FUNCTION_BLOCK FB_MotionVirtualFrame_Test EXTENDS TcUnit.FB_TestSuite
VAR
    nTestIDAssigner : INT;
    nTestID : INT := 1;
    tonTimeout : TON;
    tonStart : TON;

    stMotionStageRx : ST_MotionStage;
    stMotionStageRy : ST_MotionStage;
    stMotionStageRz : ST_MotionStage;

    stMotionStageVx : ST_MotionStage;
    stMotionStageVy : ST_MotionStage;
    stMotionStageVz : ST_MotionStage;

    fbMotionStageRx : FB_MotionStage;
    fbMotionStageRy : FB_MotionStage;
    fbMotionStageRz : FB_MotionStage;

    fbMotionStageVx : FB_MotionStage;
    fbMotionStageVy : FB_MotionStage;
    fbMotionStageVz : FB_MotionStage;

    nPositionCountsVx AT %Q* : UDINT;
    nPositionCountsVy AT %Q* : UDINT;
    nPositionCountsVz AT %Q* : UDINT;

    fbMotorTestSuite : FB_MotorTestSuite;
    fbMotionStageSetAndMoveHelper : FB_MotionStageSetAndMoveHelper;
    fbMotionStageSetHelperRx : FB_MotionStageSetHelper;
    fbMotionStageSetHelperRy : FB_MotionStageSetHelper;
    fbMotionStageSetHelperRz : FB_MotionStageSetHelper;
    fbMotionStageSetHelperVx : FB_MotionStageSetHelper;
    fbMotionStageSetHelperVy : FB_MotionStageSetHelper;
    fbMotionStageSetHelperVz : FB_MotionStageSetHelper;
    fbMotionVirtualFrame : FB_MotionVirtualFrame;
END_VAR


nTestIDAssigner := 0;

tonStart(IN := TRUE, PT := T#1s);

TestEnabled000045XYZMoveVxExpectNoErrorsCorrectPosVelAcc();

TestEnabled000090XYZMoveVxExpectNoErrorsCorrectPosVelAcc();

TestEnabled009090XYZMoveVxExpectNoErrorsCorrectPosVelAcc();

TestEnabled909090XYZMoveVxExpectNoErrorsCorrectPosVelAcc();

TestEnabledN22N21P4XYZMoveVxVyVzExpectNoErrorsCorrectPosVelAcc();

TestEnabledN22N21P4XYZMoveVyExpectNoErrorsCorrectPosVelAcc();

ACTION AssertNoErrors:

AssertFalse(
    Condition := tonTimeout.Q,
    Message := 'Timeout timer ended the test because it took longer than expected.'
);

AssertFalse(
    Condition := stMotionStageRx.bError,
    Message := 'Rx axis error detected when it should not have an error.'
);

AssertFalse(
    Condition := stMotionStageRy.bError,
    Message := 'Ry axis error detected when it should not have an error.'
);

AssertFalse(
    Condition := stMotionStageRz.bError,
    Message := 'Rz axis error detected when it should not have an error.'
);

AssertFalse(
    Condition := stMotionStageVx.bError,
    Message := 'Vx axis error detected when it should not have an error.'
);

AssertFalse(
    Condition := stMotionStageVy.bError,
    Message := 'Vy axis error detected when it should not have an error.'
);

AssertFalse(
    Condition := stMotionStageVz.bError,
    Message := 'Vz axis error detected when it should not have an error.'
);
END_ACTION


METHOD PRIVATE AssertPosVelAccCorrect
VAR_INPUT
    fDelta : LREAL;

    fRxPosExpected : LREAL;
    fRyPosExpected : LREAL;
    fRzPosExpected : LREAL;
    fVxPosExpected : LREAL;
    fVyPosExpected : LREAL;
    fVzPosExpected : LREAL;

    fRxVelExpected : LREAL;
    fRyVelExpected : LREAL;
    fRzVelExpected : LREAL;
    fVxVelExpected : LREAL;
    fVyVelExpected : LREAL;
    fVzVelExpected : LREAL;

    fRxAccExpected : LREAL;
    fRyAccExpected : LREAL;
    fRzAccExpected : LREAL;
    fVxAccExpected : LREAL;
    fVyAccExpected : LREAL;
    fVzAccExpected : LREAL;
END_VAR

// Position
AssertEquals_LREAL(
    Expected := fRxPosExpected,
    Actual := stMotionStageRx.Axis.NcToPlc.ActPos,
    Delta := fDelta,
    Message := 'Rx did not end at expected position.'
);

AssertEquals_LREAL(
    Expected := fRyPosExpected,
    Actual := stMotionStageRy.Axis.NcToPlc.ActPos,
    Delta := fDelta,
    Message := 'Ry did not end at expected position.'
);

AssertEquals_LREAL(
    Expected := fRzPosExpected,
    Actual := stMotionStageRz.Axis.NcToPlc.ActPos,
    Delta := fDelta,
    Message := 'Rz did not end at expected position.'
);

AssertEquals_LREAL(
    Expected := fVxPosExpected,
    Actual := stMotionStageVx.Axis.NcToPlc.ActPos,
    Delta := fDelta,
    Message := 'Vx did not end at expected position.'
);

AssertEquals_LREAL(
    Expected := fVyPosExpected,
    Actual := stMotionStageVy.Axis.NcToPlc.ActPos,
    Delta := fDelta,
    Message := 'Vy did not end at expected position.'
);

AssertEquals_LREAL(
    Expected := fVzPosExpected,
    Actual := stMotionStageVz.Axis.NcToPlc.ActPos,
    Delta := fDelta,
    Message := 'Vz did not end at expected position.'
);

// Velocity
AssertEquals_LREAL(
    Expected := fRxVelExpected,
    Actual := stMotionStageRx.fVelocity,
    Delta := fDelta,
    Message := 'Rx did not use the expected velocity.'
);

AssertEquals_LREAL(
    Expected := fRyVelExpected,
    Actual := stMotionStageRy.fVelocity,
    Delta := fDelta,
    Message := 'Ry did not use the expected velocity.'
);

AssertEquals_LREAL(
    Expected := fRzVelExpected,
    Actual := stMotionStageRz.fVelocity,
    Delta := fDelta,
    Message := 'Rz did not use the expected velocity.'
);

AssertEquals_LREAL(
    Expected := fVxVelExpected,
    Actual := stMotionStageVx.fVelocity,
    Delta := fDelta,
    Message := 'Vx did not use the expected velocity.'
);

AssertEquals_LREAL(
    Expected := fVyVelExpected,
    Actual := stMotionStageVy.fVelocity,
    Delta := fDelta,
    Message := 'Vy did not use the expected velocity.'
);

AssertEquals_LREAL(
    Expected := fVzVelExpected,
    Actual := stMotionStageVz.fVelocity,
    Delta := fDelta,
    Message := 'Vz did not use the expected velocity.'
);

// Acceleration
AssertEquals_LREAL(
    Expected := fRxAccExpected,
    Actual := stMotionStageRx.fAcceleration,
    Delta := fDelta,
    Message := 'Rx did not use the expected acceleration.'
);

AssertEquals_LREAL(
    Expected := fRyAccExpected,
    Actual := stMotionStageRy.fAcceleration,
    Delta := fDelta,
    Message := 'Ry did not use the expected acceleration.'
);

AssertEquals_LREAL(
    Expected := fRzAccExpected,
    Actual := stMotionStageRz.fAcceleration,
    Delta := fDelta,
    Message := 'Rz did not use the expected acceleration.'
);

AssertEquals_LREAL(
    Expected := fVxAccExpected,
    Actual := stMotionStageVx.fAcceleration,
    Delta := fDelta,
    Message := 'Vx did not use the expected acceleration.'
);

AssertEquals_LREAL(
    Expected := fVyAccExpected,
    Actual := stMotionStageVy.fAcceleration,
    Delta := fDelta,
    Message := 'Vy did not use the expected acceleration.'
);

AssertEquals_LREAL(
    Expected := fVzAccExpected,
    Actual := stMotionStageVz.fAcceleration,
    Delta := fDelta,
    Message := 'Vz did not use the expected acceleration.'
);
END_METHOD


METHOD PRIVATE InitMotors : BOOL

fbMotorTestSuite.SetEnables(stMotionStage := stMotionStageRx);
fbMotorTestSuite.SetEnables(stMotionStage := stMotionStageRy);
fbMotorTestSuite.SetEnables(stMotionStage := stMotionStageRz);
fbMotorTestSuite.SetEnables(stMotionStage := stMotionStageVx);
fbMotorTestSuite.SetEnables(stMotionStage := stMotionStageVy);
fbMotorTestSuite.SetEnables(stMotionStage := stMotionStageVz);

SetTar0();

fbMotionStageSetHelperRx(
    bExecute := TRUE,
    fStartPosition := 0.0,
    stMotionStage := stMotionStageRx,
    bResetDone => ,
    bSetDone =>
);

fbMotionStageSetHelperRy(
    bExecute := TRUE,
    fStartPosition := 0.0,
    stMotionStage := stMotionStageRy,
    bResetDone => ,
    bSetDone =>
);

fbMotionStageSetHelperRz(
    bExecute := TRUE,
    fStartPosition := 0.0,
    stMotionStage := stMotionStageRz,
    bResetDone => ,
    bSetDone =>
);

fbMotionStageSetHelperVx(
    bExecute := TRUE,
    fStartPosition := 0.0,
    stMotionStage := stMotionStageVx,
    bResetDone => ,
    bSetDone =>
);

fbMotionStageSetHelperVy(
    bExecute := TRUE,
    fStartPosition := 0.0,
    stMotionStage := stMotionStageVy,
    bResetDone => ,
    bSetDone =>
);

fbMotionStageSetHelperVz(
    bExecute := TRUE,
    fStartPosition := 0.0,
    stMotionStage := stMotionStageVz,
    bResetDone => ,
    bSetDone =>
);

IF fbMotionStageSetHelperRx.bSetDone AND
   fbMotionStageSetHelperRy.bSetDone AND
   fbMotionStageSetHelperRz.bSetDone AND
   fbMotionStageSetHelperVx.bSetDone AND
   fbMotionStageSetHelperVy.bSetDone AND
   fbMotionStageSetHelperVz.bSetDone THEN

    fbMotionStageSetHelperRx(
        bExecute := FALSE,
        fStartPosition := 0.0,
        stMotionStage := stMotionStageRx,
        bResetDone => ,
        bSetDone =>
    );

    fbMotionStageSetHelperRy(
        bExecute := FALSE,
        fStartPosition := 0.0,
        stMotionStage := stMotionStageRy,
        bResetDone => ,
        bSetDone =>
    );

    fbMotionStageSetHelperRz(
        bExecute := FALSE,
        fStartPosition := 0.0,
        stMotionStage := stMotionStageRz,
        bResetDone => ,
        bSetDone =>
    );

    fbMotionStageSetHelperVx(
        bExecute := FALSE,
        fStartPosition := 0.0,
        stMotionStage := stMotionStageVx,
        bResetDone => ,
        bSetDone =>
    );

    fbMotionStageSetHelperVy(
        bExecute := FALSE,
        fStartPosition := 0.0,
        stMotionStage := stMotionStageVy,
        bResetDone => ,
        bSetDone =>
    );

    fbMotionStageSetHelperVz(
        bExecute := FALSE,
        fStartPosition := 0.0,
        stMotionStage := stMotionStageVz,
        bResetDone => ,
        bSetDone =>
    );

    stMotionStageRx.nEnableMode := E_StageEnableMode.ALWAYS;
    stMotionStageRy.nEnableMode := E_StageEnableMode.ALWAYS;
    stMotionStageRz.nEnableMode := E_StageEnableMode.ALWAYS;
    stMotionStageVx.nEnableMode := E_StageEnableMode.ALWAYS;
    stMotionStageVy.nEnableMode := E_StageEnableMode.ALWAYS;
    stMotionStageVz.nEnableMode := E_StageEnableMode.ALWAYS;

    IF stMotionStageRx.bAllEnable AND
        stMotionStageRy.bAllEnable AND
        stMotionStageRz.bAllEnable AND
        stMotionStageVx.bAllEnable AND
        stMotionStageVy.bAllEnable AND
        stMotionStageVz.bAllEnable THEN

        InitMotors := TRUE;
    END_IF
END_IF
END_METHOD


METHOD PRIVATE SetTar0

stMotionStageVx.fPosition := 0.0;
stMotionStageVx.fVelocity := 0.0;
stMotionStageVx.fAcceleration := 0.0;

stMotionStageVy.fPosition := 0.0;
stMotionStageVy.fVelocity := 0.0;
stMotionStageVy.fAcceleration := 0.0;

stMotionStageVz.fPosition := 0.0;
stMotionStageVz.fVelocity := 0.0;
stMotionStageVz.fAcceleration := 0.0;

stMotionStageRx.fPosition := 0.0;
stMotionStageRx.fVelocity := 0.0;
stMotionStageRx.fAcceleration := 0.0;

stMotionStageRy.fPosition := 0.0;
stMotionStageRy.fVelocity := 0.0;
stMotionStageRy.fAcceleration := 0.0;

stMotionStageRz.fPosition := 0.0;
stMotionStageRz.fVelocity := 0.0;
stMotionStageRz.fAcceleration := 0.0;
END_METHOD


METHOD PRIVATE TestEnabled000045XYZMoveVxExpectNoErrorsCorrectPosVelAcc
VAR_INST
    bInit : BOOL;
    bComplete : BOOL;
    bBusyReached : BOOL;
    rtMoveCmdOnce : R_TRIG;
    fDelta : LREAL := 1e-9;
END_VAR

TEST('TestEnabled000045XYZMoveVxExpectNoErrorsCorrectPosVelAcc');

nTestIDAssigner := nTestIDAssigner + 1;

IF nTestID <> nTestIDAssigner OR NOT tonStart.Q THEN
    RETURN;
END_IF

tonTimeout(IN := TRUE, PT := T#3s);

IF NOT bInit THEN
    bInit := InitMotors();
END_IF

IF bInit THEN
    stMotionStageVx.fPosition := 15.0;
    stMotionStageVx.fVelocity := stMotionStageVx.fPosition * 2.0 / 3.0;
    stMotionStageVx.fAcceleration := stMotionStageVx.fVelocity * 5.0;
    rtMoveCmdOnce(CLK := TRUE);
    stMotionStageVx.bMoveCmd := rtMoveCmdOnce.Q;
END_IF

fbMotionVirtualFrame(
    stMotionStageRx := stMotionStageRx,
    stMotionStageRy := stMotionStageRy,
    stMotionStageRz := stMotionStageRz,
    stMotionStageVx := stMotionStageVx,
    stMotionStageVy := stMotionStageVy,
    stMotionStageVz := stMotionStageVz,
    bEnable := TRUE,
    fAlphaDegrees := 0.0,
    fBetaDegrees := 0.0,
    fGammaDegrees := 45.0,
    sOrder := 'XYZ',
    bBaseToNew := TRUE,
    fbVirtActPositionVec3 => ,
    fbVirtActVelocityVec3 => ,
    fbVirtActAcceleraVec3 =>
);

IF stMotionStageVx.bBusy THEN
    bBusyReached := TRUE;
END_IF

IF bBusyReached AND NOT stMotionStageVx.bBusy THEN
    bComplete := TRUE;
END_IF

IF (bComplete AND
    NOT stMotionStageVx.bBusy AND
    NOT stMotionStageVy.bBusy AND
    NOT stMotionStageVz.bBusy AND
    NOT stMotionStageRx.bBusy AND
    NOT stMotionStageRy.bBusy AND
    NOT stMotionStageRz.bBusy)
    OR tonTimeout.Q THEN

    AssertNoErrors();

    AssertPosVelAccCorrect(
        fDelta := fDelta,
        fRxPosExpected := stMotionStageVx.fPosition * SQRT(2.0) / 2.0,
        fRyPosExpected := stMotionStageVx.fPosition * SQRT(2.0) / 2.0,
        fRzPosExpected := 0.0,
        fVxPosExpected := stMotionStageVx.fPosition,
        fVyPosExpected := 0.0,
        fVzPosExpected := 0.0,
        fRxVelExpected := stMotionStageVx.fVelocity * SQRT(2.0) / 2.0,
        fRyVelExpected := stMotionStageVx.fVelocity * SQRT(2.0) / 2.0,
        fRzVelExpected := 0.0,
        fVxVelExpected := stMotionStageVx.fVelocity,
        fVyVelExpected := 0.0,
        fVzVelExpected := 0.0,
        fRxAccExpected := stMotionStageVx.fAcceleration * SQRT(2.0) / 2.0,
        fRyAccExpected := stMotionStageVx.fAcceleration * SQRT(2.0) / 2.0,
        fRzAccExpected := 0.0,
        fVxAccExpected := stMotionStageVx.fAcceleration,
        fVyAccExpected := 0.0,
        fVzAccExpected := 0.0
    );

    TEST_FINISHED();

    tonTimeout(IN := FALSE);

    nTestID := nTestID + 1;
END_IF

fbMotionStageRx(stMotionStage := stMotionStageRx);
fbMotionStageRy(stMotionStage := stMotionStageRy);
fbMotionStageRz(stMotionStage := stMotionStageRz);

fbMotionStageVx(stMotionStage := stMotionStageVx);
fbMotionStageVy(stMotionStage := stMotionStageVy);
fbMotionStageVz(stMotionStage := stMotionStageVz);

nPositionCountsVx := LREAL_TO_UDINT((fbMotionVirtualFrame.fbVirtActPositionVec3.x + 100.0) * 1e6);
nPositionCountsVy := LREAL_TO_UDINT((fbMotionVirtualFrame.fbVirtActPositionVec3.y + 100.0) * 1e6);
nPositionCountsVz := LREAL_TO_UDINT((fbMotionVirtualFrame.fbVirtActPositionVec3.z + 100.0) * 1e6);
END_METHOD


METHOD PRIVATE TestEnabled000090XYZMoveVxExpectNoErrorsCorrectPosVelAcc
VAR_INST
    bInit : BOOL;
    bComplete : BOOL;
    bBusyReached : BOOL;
    rtMoveCmdOnce : R_TRIG;
    fDelta : LREAL := 1e-9;
END_VAR

TEST('TestEnabled000090XYZMoveVxExpectNoErrorsCorrectPosVelAcc');

nTestIDAssigner := nTestIDAssigner + 1;

IF nTestID <> nTestIDAssigner OR NOT tonStart.Q THEN
    RETURN;
END_IF

tonTimeout(IN := TRUE, PT := T#3s);

IF NOT bInit THEN
    bInit := InitMotors();
END_IF

IF bInit THEN
    stMotionStageVx.fPosition := 20.0;
    stMotionStageVx.fVelocity := stMotionStageVx.fPosition * 2.0 / 3.0;
    stMotionStageVx.fAcceleration := stMotionStageVx.fVelocity * 5.0;
    rtMoveCmdOnce(CLK := TRUE);
    stMotionStageVx.bMoveCmd := rtMoveCmdOnce.Q;
END_IF

fbMotionVirtualFrame(
    stMotionStageRx := stMotionStageRx,
    stMotionStageRy := stMotionStageRy,
    stMotionStageRz := stMotionStageRz,
    stMotionStageVx := stMotionStageVx,
    stMotionStageVy := stMotionStageVy,
    stMotionStageVz := stMotionStageVz,
    bEnable := TRUE,
    fAlphaDegrees := 0.0,
    fBetaDegrees := 0.0,
    fGammaDegrees := 90.0,
    sOrder := 'XYZ',
    bBaseToNew := TRUE,
    fbVirtActPositionVec3 => ,
    fbVirtActVelocityVec3 => ,
    fbVirtActAcceleraVec3 =>
);

IF stMotionStageVx.bBusy THEN
    bBusyReached := TRUE;
END_IF

IF bBusyReached AND NOT stMotionStageVx.bBusy THEN
    bComplete := TRUE;
END_IF

IF (bComplete AND
    NOT stMotionStageVx.bBusy AND
    NOT stMotionStageVy.bBusy AND
    NOT stMotionStageVz.bBusy AND
    NOT stMotionStageRx.bBusy AND
    NOT stMotionStageRy.bBusy AND
    NOT stMotionStageRz.bBusy)
    OR tonTimeout.Q THEN

    AssertNoErrors();

    AssertPosVelAccCorrect(
        fDelta := fDelta,
        fRxPosExpected := 0.0,
        fRyPosExpected := stMotionStageVx.fPosition,
        fRzPosExpected := 0.0,
        fVxPosExpected := stMotionStageVx.fPosition,
        fVyPosExpected := 0.0,
        fVzPosExpected := 0.0,
        fRxVelExpected := 0.0,
        fRyVelExpected := stMotionStageVx.fVelocity,
        fRzVelExpected := 0.0,
        fVxVelExpected := stMotionStageVx.fVelocity,
        fVyVelExpected := 0.0,
        fVzVelExpected := 0.0,
        fRxAccExpected := 0.0,
        fRyAccExpected := stMotionStageVx.fAcceleration,
        fRzAccExpected := 0.0,
        fVxAccExpected := stMotionStageVx.fAcceleration,
        fVyAccExpected := 0.0,
        fVzAccExpected := 0.0
    );

    TEST_FINISHED();

    tonTimeout(IN := FALSE);

    nTestID := nTestID + 1;
END_IF

fbMotionStageRx(stMotionStage := stMotionStageRx);
fbMotionStageRy(stMotionStage := stMotionStageRy);
fbMotionStageRz(stMotionStage := stMotionStageRz);

fbMotionStageVx(stMotionStage := stMotionStageVx);
fbMotionStageVy(stMotionStage := stMotionStageVy);
fbMotionStageVz(stMotionStage := stMotionStageVz);

nPositionCountsVx := LREAL_TO_UDINT((fbMotionVirtualFrame.fbVirtActPositionVec3.x + 100.0) * 1e6);
nPositionCountsVy := LREAL_TO_UDINT((fbMotionVirtualFrame.fbVirtActPositionVec3.y + 100.0) * 1e6);
nPositionCountsVz := LREAL_TO_UDINT((fbMotionVirtualFrame.fbVirtActPositionVec3.z + 100.0) * 1e6);
END_METHOD


METHOD PRIVATE TestEnabled009090XYZMoveVxExpectNoErrorsCorrectPosVelAcc
VAR_INST
    bInit : BOOL;
    bComplete : BOOL;
    bBusyReached : BOOL;
    rtMoveCmdOnce : R_TRIG;
    fDelta : LREAL := 1e-9;
END_VAR

TEST('TestEnabled009090XYZMoveVxExpectNoErrorsCorrectPosVelAcc');

nTestIDAssigner := nTestIDAssigner + 1;

IF nTestID <> nTestIDAssigner OR NOT tonStart.Q THEN
    RETURN;
END_IF

tonTimeout(IN := TRUE, PT := T#3s);

IF NOT bInit THEN
    bInit := InitMotors();
END_IF

IF bInit THEN
    stMotionStageVx.fPosition := 25.0;
    stMotionStageVx.fVelocity := stMotionStageVx.fPosition * 2.0 / 3.0;
    stMotionStageVx.fAcceleration := stMotionStageVx.fVelocity * 5.0;
    rtMoveCmdOnce(CLK := TRUE);
    stMotionStageVx.bMoveCmd := rtMoveCmdOnce.Q;
END_IF

fbMotionVirtualFrame(
    stMotionStageRx := stMotionStageRx,
    stMotionStageRy := stMotionStageRy,
    stMotionStageRz := stMotionStageRz,
    stMotionStageVx := stMotionStageVx,
    stMotionStageVy := stMotionStageVy,
    stMotionStageVz := stMotionStageVz,
    bEnable := TRUE,
    fAlphaDegrees := 0.0,
    fBetaDegrees := 90.0,
    fGammaDegrees := 90.0,
    sOrder := 'XYZ',
    bBaseToNew := TRUE,
    fbVirtActPositionVec3 => ,
    fbVirtActVelocityVec3 => ,
    fbVirtActAcceleraVec3 =>
);

IF stMotionStageVx.bBusy THEN
    bBusyReached := TRUE;
END_IF

IF bBusyReached AND NOT stMotionStageVx.bBusy THEN
    bComplete := TRUE;
END_IF

IF (bComplete AND
    NOT stMotionStageVx.bBusy AND
    NOT stMotionStageVy.bBusy AND
    NOT stMotionStageVz.bBusy AND
    NOT stMotionStageRx.bBusy AND
    NOT stMotionStageRy.bBusy AND
    NOT stMotionStageRz.bBusy)
    OR tonTimeout.Q THEN

    AssertNoErrors();

    AssertPosVelAccCorrect(
        fDelta := fDelta,
        fRxPosExpected := 0.0,
        fRyPosExpected := stMotionStageVx.fPosition,
        fRzPosExpected := 0.0,
        fVxPosExpected := stMotionStageVx.fPosition,
        fVyPosExpected := 0.0,
        fVzPosExpected := 0.0,
        fRxVelExpected := 0.0,
        fRyVelExpected := stMotionStageVx.fVelocity,
        fRzVelExpected := 0.0,
        fVxVelExpected := stMotionStageVx.fVelocity,
        fVyVelExpected := 0.0,
        fVzVelExpected := 0.0,
        fRxAccExpected := 0.0,
        fRyAccExpected := stMotionStageVx.fAcceleration,
        fRzAccExpected := 0.0,
        fVxAccExpected := stMotionStageVx.fAcceleration,
        fVyAccExpected := 0.0,
        fVzAccExpected := 0.0
    );

    TEST_FINISHED();

    tonTimeout(IN := FALSE);

    nTestID := nTestID + 1;
END_IF

fbMotionStageRx(stMotionStage := stMotionStageRx);
fbMotionStageRy(stMotionStage := stMotionStageRy);
fbMotionStageRz(stMotionStage := stMotionStageRz);

fbMotionStageVx(stMotionStage := stMotionStageVx);
fbMotionStageVy(stMotionStage := stMotionStageVy);
fbMotionStageVz(stMotionStage := stMotionStageVz);

nPositionCountsVx := LREAL_TO_UDINT((fbMotionVirtualFrame.fbVirtActPositionVec3.x + 100.0) * 1e6);
nPositionCountsVy := LREAL_TO_UDINT((fbMotionVirtualFrame.fbVirtActPositionVec3.y + 100.0) * 1e6);
nPositionCountsVz := LREAL_TO_UDINT((fbMotionVirtualFrame.fbVirtActPositionVec3.z + 100.0) * 1e6);
END_METHOD


METHOD PRIVATE TestEnabled909090XYZMoveVxExpectNoErrorsCorrectPosVelAcc
VAR_INST
    bInit : BOOL;
    bComplete : BOOL;
    bBusyReached : BOOL;
    rtMoveCmdOnce : R_TRIG;
    fDelta : LREAL := 1e-9;
END_VAR

TEST('TestEnabled909090XYZMoveVxExpectNoErrorsCorrectPosVelAcc');

nTestIDAssigner := nTestIDAssigner + 1;

IF nTestID <> nTestIDAssigner OR NOT tonStart.Q THEN
    RETURN;
END_IF

tonTimeout(IN := TRUE, PT := T#3s);

IF NOT bInit THEN
    bInit := InitMotors();
END_IF

IF bInit THEN
    stMotionStageVx.fPosition := 35.0;
    stMotionStageVx.fVelocity := stMotionStageVx.fPosition * 2.0 / 3.0;
    stMotionStageVx.fAcceleration := stMotionStageVx.fVelocity * 5.0;
    rtMoveCmdOnce(CLK := TRUE);
    stMotionStageVx.bMoveCmd := rtMoveCmdOnce.Q;
END_IF

fbMotionVirtualFrame(
    stMotionStageRx := stMotionStageRx,
    stMotionStageRy := stMotionStageRy,
    stMotionStageRz := stMotionStageRz,
    stMotionStageVx := stMotionStageVx,
    stMotionStageVy := stMotionStageVy,
    stMotionStageVz := stMotionStageVz,
    bEnable := TRUE,
    fAlphaDegrees := 90.0,
    fBetaDegrees := 90.0,
    fGammaDegrees := 90.0,
    sOrder := 'XYZ',
    bBaseToNew := TRUE,
    fbVirtActPositionVec3 => ,
    fbVirtActVelocityVec3 => ,
    fbVirtActAcceleraVec3 =>
);

IF stMotionStageVx.bBusy THEN
    bBusyReached := TRUE;
END_IF

IF bBusyReached AND NOT stMotionStageVx.bBusy THEN
    bComplete := TRUE;
END_IF

IF (bComplete AND
    NOT stMotionStageVx.bBusy AND
    NOT stMotionStageVy.bBusy AND
    NOT stMotionStageVz.bBusy AND
    NOT stMotionStageRx.bBusy AND
    NOT stMotionStageRy.bBusy AND
    NOT stMotionStageRz.bBusy)
    OR tonTimeout.Q THEN

    AssertNoErrors();

    AssertPosVelAccCorrect(
        fDelta := fDelta,
        fRxPosExpected := 0.0,
        fRyPosExpected := 0.0,
        fRzPosExpected := stMotionStageVx.fPosition,
        fVxPosExpected := stMotionStageVx.fPosition,
        fVyPosExpected := 0.0,
        fVzPosExpected := 0.0,
        fRxVelExpected := 0.0,
        fRyVelExpected := 0.0,
        fRzVelExpected := stMotionStageVx.fVelocity,
        fVxVelExpected := stMotionStageVx.fVelocity,
        fVyVelExpected := 0.0,
        fVzVelExpected := 0.0,
        fRxAccExpected := 0.0,
        fRyAccExpected := 0.0,
        fRzAccExpected := stMotionStageVx.fAcceleration,
        fVxAccExpected := stMotionStageVx.fAcceleration,
        fVyAccExpected := 0.0,
        fVzAccExpected := 0.0
    );

    TEST_FINISHED();

    tonTimeout(IN := FALSE);

    nTestID := nTestID + 1;
END_IF

fbMotionStageRx(stMotionStage := stMotionStageRx);
fbMotionStageRy(stMotionStage := stMotionStageRy);
fbMotionStageRz(stMotionStage := stMotionStageRz);

fbMotionStageVx(stMotionStage := stMotionStageVx);
fbMotionStageVy(stMotionStage := stMotionStageVy);
fbMotionStageVz(stMotionStage := stMotionStageVz);

nPositionCountsVx := LREAL_TO_UDINT((fbMotionVirtualFrame.fbVirtActPositionVec3.x + 100.0) * 1e6);
nPositionCountsVy := LREAL_TO_UDINT((fbMotionVirtualFrame.fbVirtActPositionVec3.y + 100.0) * 1e6);
nPositionCountsVz := LREAL_TO_UDINT((fbMotionVirtualFrame.fbVirtActPositionVec3.z + 100.0) * 1e6);
END_METHOD


METHOD PRIVATE TestEnabledN22N21P4XYZMoveVxVyVzExpectNoErrorsCorrectPosVelAcc
VAR_INST
    bInit : BOOL;
    bComplete : BOOL;
    bBusyReached : BOOL;
    rtMoveCmdOnce : R_TRIG;
    fDelta : LREAL := 1e-9;
END_VAR

TEST('TestEnabledN22N21P4XYZMoveVxVyVzExpectNoErrorsCorrectPosVelAcc');

nTestIDAssigner := nTestIDAssigner + 1;

IF nTestID <> nTestIDAssigner OR NOT tonStart.Q THEN
    RETURN;
END_IF

tonTimeout(IN := TRUE, PT := T#3s);

IF NOT bInit THEN
    bInit := InitMotors();
END_IF

IF bInit THEN
    rtMoveCmdOnce(CLK := TRUE);

    stMotionStageVx.fPosition := 15.0;
    stMotionStageVx.fVelocity := stMotionStageVx.fPosition * 2.0 / 3.0;
    stMotionStageVx.fAcceleration := stMotionStageVx.fVelocity * 5.0;
    stMotionStageVx.bMoveCmd := rtMoveCmdOnce.Q;

    stMotionStageVy.fPosition := -30.0;
    stMotionStageVy.fVelocity := ABS(stMotionStageVy.fPosition * 2.0 / 3.0);
    stMotionStageVy.fAcceleration := ABS(stMotionStageVy.fVelocity * 5.0);
    stMotionStageVy.bMoveCmd := rtMoveCmdOnce.Q;

    stMotionStageVz.fPosition := 45.0;
    stMotionStageVz.fVelocity := stMotionStageVz.fPosition * 2.0 / 3.0;
    stMotionStageVz.fAcceleration := stMotionStageVz.fVelocity * 5.0;
    stMotionStageVz.bMoveCmd := rtMoveCmdOnce.Q;
END_IF

fbMotionVirtualFrame(
    stMotionStageRx := stMotionStageRx,
    stMotionStageRy := stMotionStageRy,
    stMotionStageRz := stMotionStageRz,
    stMotionStageVx := stMotionStageVx,
    stMotionStageVy := stMotionStageVy,
    stMotionStageVz := stMotionStageVz,
    bEnable := TRUE,
    fAlphaDegrees := -22.21,
    fBetaDegrees := -20.7,
    fGammaDegrees := 3.793,
    sOrder := 'XYZ',
    bBaseToNew := FALSE,
    fbVirtActPositionVec3 => ,
    fbVirtActVelocityVec3 => ,
    fbVirtActAcceleraVec3 =>
);

IF stMotionStageVx.bBusy AND stMotionStageVy.bBusy AND stMotionStageVz.bBusy THEN
    bBusyReached := TRUE;
END_IF

IF bBusyReached AND NOT stMotionStageVx.bBusy AND NOT stMotionStageVy.bBusy AND NOT stMotionStageVz.bBusy THEN
    bComplete := TRUE;
END_IF

IF (bComplete AND
    NOT stMotionStageVx.bBusy AND
    NOT stMotionStageVy.bBusy AND
    NOT stMotionStageVz.bBusy AND
    NOT stMotionStageRx.bBusy AND
    NOT stMotionStageRy.bBusy AND
    NOT stMotionStageRz.bBusy)
    OR tonTimeout.Q THEN

    AssertNoErrors();

    AssertPosVelAccCorrect(
        fDelta := fDelta,
        fRxPosExpected := 21.732640182123049,
        fRyPosExpected := -46.323371856381527,
        fRzPosExpected := 23.061603816078627,
        fVxPosExpected := stMotionStageVx.fPosition,
        fVyPosExpected := stMotionStageVy.fPosition,
        fVzPosExpected := stMotionStageVz.fPosition,
        fRxVelExpected := 14.488426788082032,
        fRyVelExpected := 30.882247904254346,
        fRzVelExpected := 15.374402544052412,
        fVxVelExpected := stMotionStageVx.fVelocity,
        fVyVelExpected := stMotionStageVy.fVelocity,
        fVzVelExpected := stMotionStageVz.fVelocity,
        fRxAccExpected := 0.724421339404102 * 1e2,
        fRyAccExpected := 1.544112395212718 * 1e2,
        fRzAccExpected := 0.768720127202621 * 1e2,
        fVxAccExpected := stMotionStageVx.fAcceleration,
        fVyAccExpected := stMotionStageVy.fAcceleration,
        fVzAccExpected := stMotionStageVz.fAcceleration
    );

    TEST_FINISHED();

    tonTimeout(IN := FALSE);

    nTestID := nTestID + 1;
END_IF

fbMotionStageRx(stMotionStage := stMotionStageRx);
fbMotionStageRy(stMotionStage := stMotionStageRy);
fbMotionStageRz(stMotionStage := stMotionStageRz);

fbMotionStageVx(stMotionStage := stMotionStageVx);
fbMotionStageVy(stMotionStage := stMotionStageVy);
fbMotionStageVz(stMotionStage := stMotionStageVz);

nPositionCountsVx := LREAL_TO_UDINT((fbMotionVirtualFrame.fbVirtActPositionVec3.x + 100.0) * 1e6);
nPositionCountsVy := LREAL_TO_UDINT((fbMotionVirtualFrame.fbVirtActPositionVec3.y + 100.0) * 1e6);
nPositionCountsVz := LREAL_TO_UDINT((fbMotionVirtualFrame.fbVirtActPositionVec3.z + 100.0) * 1e6);
END_METHOD


METHOD PRIVATE TestEnabledN22N21P4XYZMoveVyExpectNoErrorsCorrectPosVelAcc
VAR_INST
    bInit : BOOL;
    bComplete : BOOL;
    bBusyReached : BOOL;
    rtMoveCmdOnce : R_TRIG;
    fDelta : LREAL := 1e-9;
END_VAR

TEST('TestEnabledN22N21P4XYZMoveVyExpectNoErrorsCorrectPosVelAcc');

nTestIDAssigner := nTestIDAssigner + 1;

IF nTestID <> nTestIDAssigner OR NOT tonStart.Q THEN
    RETURN;
END_IF

tonTimeout(IN := TRUE, PT := T#3s);

IF NOT bInit THEN
    bInit := InitMotors();
END_IF

IF bInit THEN
    stMotionStageVy.fPosition := 30.0;
    stMotionStageVy.fVelocity := stMotionStageVy.fPosition * 2.0 / 3.0;
    stMotionStageVy.fAcceleration := stMotionStageVy.fVelocity * 5.0;
    rtMoveCmdOnce(CLK := TRUE);
    stMotionStageVy.bMoveCmd := rtMoveCmdOnce.Q;
END_IF

fbMotionVirtualFrame(
    stMotionStageRx := stMotionStageRx,
    stMotionStageRy := stMotionStageRy,
    stMotionStageRz := stMotionStageRz,
    stMotionStageVx := stMotionStageVx,
    stMotionStageVy := stMotionStageVy,
    stMotionStageVz := stMotionStageVz,
    bEnable := TRUE,
    fAlphaDegrees := -22.21,
    fBetaDegrees := -20.7,
    fGammaDegrees := 3.793,
    sOrder := 'XYZ',
    bBaseToNew := FALSE,
    fbVirtActPositionVec3 => ,
    fbVirtActVelocityVec3 => ,
    fbVirtActAcceleraVec3 =>
);

IF stMotionStageVy.bBusy THEN
    bBusyReached := TRUE;
END_IF

IF bBusyReached AND NOT stMotionStageVy.bBusy THEN
    bComplete := TRUE;
END_IF

IF (bComplete AND
    NOT stMotionStageVx.bBusy AND
    NOT stMotionStageVy.bBusy AND
    NOT stMotionStageVz.bBusy AND
    NOT stMotionStageRx.bBusy AND
    NOT stMotionStageRy.bBusy AND
    NOT stMotionStageRz.bBusy)
    OR tonTimeout.Q THEN

    AssertNoErrors();

    AssertPosVelAccCorrect(
        fDelta := fDelta,
        fRxPosExpected := 5.836964390001455,
        fRyPosExpected := 27.448135465863341,
        fRzPosExpected := 10.608001987060069,
        fVxPosExpected := 0.0,
        fVyPosExpected := stMotionStageVy.fPosition,
        fVzPosExpected := 0.0,
        fRxVelExpected := 5.836964390001455 * 2.0 / 3.0,
        fRyVelExpected := 27.448135465863341 * 2.0 / 3.0,
        fRzVelExpected := 10.608001987060069 * 2.0 / 3.0,
        fVxVelExpected := 0.0,
        fVyVelExpected := stMotionStageVy.fVelocity,
        fVzVelExpected := 0.0,
        fRxAccExpected := 5.836964390001455 * 2.0 / 3.0 * 5.0,
        fRyAccExpected := 27.448135465863341 * 2.0 / 3.0 * 5.0,
        fRzAccExpected := 10.608001987060069 * 2.0 / 3.0 * 5.0,
        fVxAccExpected := 0.0,
        fVyAccExpected := stMotionStageVy.fAcceleration,
        fVzAccExpected := 0.0
    );

    TEST_FINISHED();

    tonTimeout(IN := FALSE);

    nTestID := nTestID + 1;
END_IF

fbMotionStageRx(stMotionStage := stMotionStageRx);
fbMotionStageRy(stMotionStage := stMotionStageRy);
fbMotionStageRz(stMotionStage := stMotionStageRz);

fbMotionStageVx(stMotionStage := stMotionStageVx);
fbMotionStageVy(stMotionStage := stMotionStageVy);
fbMotionStageVz(stMotionStage := stMotionStageVz);

nPositionCountsVx := LREAL_TO_UDINT((fbMotionVirtualFrame.fbVirtActPositionVec3.x + 100.0) * 1e6);
nPositionCountsVy := LREAL_TO_UDINT((fbMotionVirtualFrame.fbVirtActPositionVec3.y + 100.0) * 1e6);
nPositionCountsVz := LREAL_TO_UDINT((fbMotionVirtualFrame.fbVirtActPositionVec3.z + 100.0) * 1e6);
END_METHOD

END_FUNCTION_BLOCK

(* stored: Version 1.1.0.1
   POU FB_MotionVirtualFrame_Test: Id {89c3fcc0-8932-48a8-9976-db5e1ce2e9c1}, SpecialFunc None
   Action AssertNoErrors: Id {835be31f-8489-492c-bbc8-90f1a0c04eb1}
   Method AssertPosVelAccCorrect: Id {645a18f6-30c6-4966-a4ea-a55c7fe24cdb}
   Method InitMotors: Id {62a5dad0-d7c7-4660-a2ba-05b951ff6ec0}
   Method SetTar0: Id {46f058f5-eb38-4947-8a98-e9788bc7e851}
   Method TestEnabled000045XYZMoveVxExpectNoErrorsCorrectPosVelAcc: Id {2d40004f-479b-4cbc-9e82-633d171550b1}
   Method TestEnabled000090XYZMoveVxExpectNoErrorsCorrectPosVelAcc: Id {96619493-4949-4dca-ad6e-5a7f16038b00}
   Method TestEnabled009090XYZMoveVxExpectNoErrorsCorrectPosVelAcc: Id {1e6baa8a-c190-4123-9357-8013455bb605}
   Method TestEnabled909090XYZMoveVxExpectNoErrorsCorrectPosVelAcc: Id {6c8e3a8e-65f7-4fff-beca-5b108daa78c7}
   Method TestEnabledN22N21P4XYZMoveVxVyVzExpectNoErrorsCorrectPosVelAcc: Id {346202be-906d-4ffe-aa6d-c53059f69711}
   Method TestEnabledN22N21P4XYZMoveVyExpectNoErrorsCorrectPosVelAcc: Id {21051135-eac8-427d-b480-287c40f7c624} *)
